FUNCTION_BLOCK EL4114
VAR
	_io : EL4xx4_Data;
	{attribute addProperty Name "WcState"}
	_wcState : WcStateBase;
	{attribute addProperty Name "Info data"}
	_infoData : InfoDataAds;
END_VAR

PROPERTY IO : REFERENCE TO EL4xx4_Data
GET
IO REF= _io;
END_GET
END_PROPERTY

PROPERTY WcState : REFERENCE TO WcStateBase
GET
WcState REF= _wcState;
END_GET
END_PROPERTY

END_FUNCTION_BLOCK

(* stored: Version 1.1.0.1, ProductVersion 3.1.4024.9
   POU EL4114: Id {3e0fbf20-8334-09f6-392e-0ac19e5fe2e4}, SpecialFunc None
   Property IO: Id {e036298f-1c51-0f4e-22c0-1c6aac635716}
   Get Get: Id {ce44b9b9-3333-0706-0717-9983cf496de5}
   Property WcState: Id {411319bd-1bca-0e9c-1190-c0c4e6fc66d8}
   Get Get: Id {1422cad9-397a-0347-2fe4-7c28b3518eae} *)
